# EPICS autosave request: iocBoot/sioc-in10-im01/sioc-in10-im01.req
file "facet2.req" AREA=IN10,POS=431
file "facet2.req" AREA=IN10,POS=591
